FUNCTION_BLOCK FB_EventLogger
VAR
	eventBuffer: ARRAY[1..EVENT_BUFFER_SIZE] OF ST_Event;
	currentBufferIndex: USINT := 0;
	
	_eventStorage: EventStorage; // setting this in the constructor/FB_init
	
END_VAR
VAR CONSTANT
	EVENT_BUFFER_SIZE: INT := 10;
END_VAR

METHOD AddEvent : BOOL
VAR_INPUT
	event: ST_EVENT;
END_VAR
IF (currentBufferIndex + 1) < EVENT_BUFFER_SIZE THEN
	currentBufferIndex := currentBufferIndex + 1;
	F_UpdateEventTimeStamp(st_event := event);
	event.nEventId := currentBufferIndex;
	eventBuffer[currentBufferIndex]:= event;
	
	// Here we store event persistently
	_eventStorage.StoreEvent(st_event:= event);
END_IF
END_METHOD

(****
 
Called implicitly whenever an instance of the Event Logger is instantiated.
Like a Constructor.

*****)

METHOD FB_init : BOOL
VAR_INPUT
	bInitRetains : BOOL; // if TRUE, the retain variables are initialized (warm start / cold start)
	bInCopyCode : BOOL;  // if TRUE, the instance afterwards gets moved into the copy code (online change)

	// Require something that implementes EventStorage interface	
	eventStorage: EventStorage;
	
END_VAR
_eventStorage := eventStorage;
END_METHOD

END_FUNCTION_BLOCK

(* stored: Version 1.1.0.1, ProductVersion 3.1.4024.12
   POU FB_EventLogger: Id {a942f2bf-159f-4cae-ba24-c9efa6a07217}, SpecialFunc None
   Method AddEvent: Id {1c250104-f2e5-40ae-8808-3208892b77db}
   Method FB_init: Id {d8743572-4575-42a7-aef9-69c0c0f25234} *)
